INTERFACE I_Drive

METHOD AutoLedOff : BOOL
VAR_INPUT
END_VAR
END_METHOD

METHOD AutoLedOn : BOOL
VAR_INPUT
END_VAR
END_METHOD

METHOD SwitchOff : BOOL
VAR_INPUT
END_VAR
END_METHOD

METHOD SwitchOn : BOOL
VAR_INPUT
END_VAR
END_METHOD

METHOD WorkCounterOff : BOOL
VAR_INPUT
END_VAR
END_METHOD

METHOD WorkCounterOn : BOOL
VAR_INPUT
END_VAR
END_METHOD

END_INTERFACE

(* stored: Version 1.1.0.1, ProductVersion 3.1.4024.12
   Itf I_Drive: Id {32f04a35-7cc4-4a82-a219-6ae04a30264f}
   Method AutoLedOff: Id {9d5a9030-3dfb-40e3-8783-1389ac006255}
   Method AutoLedOn: Id {93a30ca8-66d3-41a8-95b1-10347e5c84ce}
   Method SwitchOff: Id {ae9140d4-60e7-4ab0-9aba-6c098fbeaf6c}
   Method SwitchOn: Id {99be391c-6b6f-45b3-9fbc-71b1518bbbdd}
   Method WorkCounterOff: Id {2aa25d40-acd0-47fc-a6de-f1a52539585e}
   Method WorkCounterOn: Id {d4898fdc-7a8e-4e01-92c3-0f762b05b316} *)
